PROGRAM MAIN
VAR
	axisX, axisY : AXIS_REF;
	diX, diY AT %I* : BOOL;
	bEnable : BOOL;
	powerX, powerY : MC_Power;
	resetX, resetY : MC_Reset;
	homeX, homeY : MC_Home;
	moveAbsY, moveAbsY : MC_MoveAbsolute;
END_VAR

END_PROGRAM

(* stored: Version 1.1.0.1, ProductVersion 3.1.0.26
   POU MAIN: Id {921adec3-9538-4142-a9cc-7f60e269c50c} *)
